FUNCTION_BLOCK ABSTRACT LaserBase EXTENDS TExecution IMPLEMENTS IDevice
VAR_INPUT
END_VAR
VAR_OUTPUT
END_VAR
VAR
	{attribute 'OPC.UA.DA' := '0'}
	_name : STRING;
	{attribute 'OPC.UA.DA' := '0'}
	_deviceID : STRING;				
	{attribute 'OPC.UA.DA' := '0'}	
	_family : DeviceFamily;	
	{attribute 'OPC.UA.DA' := '0'}
	_logger : Logger;
	{attribute 'OPC.UA.DA' := '0'}
	_message : StringBuilder;
	{attribute 'OPC.UA.DA' := '0'}
	_laserConfig : DeviceConfiguration;	
END_VAR

PROPERTY DeviceID : STRING
GET
DeviceID := _deviceID;
END_GET
SET
_deviceID := DeviceID;
END_SET
END_PROPERTY

PROPERTY Family : DeviceFamily
GET
Family := _family;
END_GET
SET
_family := Family;
END_SET
END_PROPERTY

METHOD PROTECTED ABSTRACT GetInterlockStatus 
VAR_INPUT
END_VAR
END_METHOD

PROPERTY Name : STRING
GET
Name := _name;
END_GET
SET
_name := Name;
END_SET
END_PROPERTY

METHOD PROTECTED ABSTRACT PowerOff
VAR_INPUT
	Execute : BOOL;
END_VAR
END_METHOD

METHOD PROTECTED ABSTRACT PowerOn
VAR_INPUT
	Execute : BOOL;
END_VAR
END_METHOD

METHOD PROTECTED ABSTRACT ReadPower 
VAR_INPUT
END_VAR
END_METHOD

METHOD PROTECTED ABSTRACT SetPower
VAR_INPUT
	Execute : BOOL;
	Power : LREAL;
END_VAR
END_METHOD

END_FUNCTION_BLOCK

(* stored: Version 1.1.0.1, ProductVersion 3.1.4024.12
   POU LaserBase: Id {c5bc4fb2-2b01-480f-a0fe-01264f28b56a}, SpecialFunc None
   Property DeviceID: Id {6a7f319d-17fc-4921-92c7-304c515b8418}
   Get Get: Id {cee97da2-36f1-43c2-9ea4-531df3a00e84}
   Set Set: Id {4e7a1184-631d-4b8e-b549-03609fbd4df2}
   Property Family: Id {0bebef37-aac3-4176-9317-4fa592bcbde9}
   Get Get: Id {7d88df11-65a0-4b9f-9248-89207ed8226d}
   Set Set: Id {f0916c8c-215f-41c6-9818-1a789bd6b13f}
   Method GetInterlockStatus: Id {f39e805d-c69a-4a4c-b062-44a2b433cf86}
   Property Name: Id {324bb144-2c14-4489-a92f-3b0f1c962321}
   Get Get: Id {bfc52385-d343-48cf-be00-93a8daf5ca4b}
   Set Set: Id {db3bd38c-3494-48ea-a27d-42314e8824da}
   Method PowerOff: Id {9593aedd-dcaa-487e-af79-88d78b8509f7}
   Method PowerOn: Id {e5c2506d-efa7-4153-8c58-5ffd70314b7c}
   Method ReadPower: Id {1f5a33c0-da1a-4dd7-98c7-c14455db8601}
   Method SetPower: Id {9c1220b2-e20d-45d9-adf4-94f08793949c} *)
